ABB RAPID module: CalibData.modx

MODULE CalibData
    TASK PERS tooldata SpreaderEOT:=[TRUE,[[0,0,150],[0.707106783,0.000000004,-0.000000001,-0.70710678]],[1,[0,0,1],[1,0,0,0],0,0,0]];
    TASK PERS wobjdata Wall:=[FALSE,TRUE,"",[[0,0,0],[1,0,0,0]],[[1000.052,350,860.843],[0.5,-0.5,0.5,-0.5]]];
ENDMODULE
